TYPE ST_Steuerung_auto_manu_opti_REAL :
STRUCT
	auto			: REAL;
	manu			: REAL;
	manu_Modus		: BOOL;
	opti			: REAL;
	opti_Modus		: BOOL;
END_STRUCT
END_TYPE

(* stored: Version 1.1.0.1, ProductVersion 3.1.4024.9
   DUT ST_Steuerung_auto_manu_opti_REAL: Id {cead52d4-8a98-454f-b7ec-ce1ca5127b54} *)
